FUNCTION_BLOCK TcoDigitalSensor EXTENDS TcoCore.TcoComponent
VAR_IN_OUT
	inoSignal : BOOL;
END_VAR

VAR
	_signal : BOOL;
	_adr : ULINT;
END_VAR

IF(__ISVALIDREF(inoSignal)) THEN
	_signal := inoSignal;
	_adr := ADR(inoSignal);
END_IF;

METHOD FB_init : BOOL
VAR_INPUT
	bInitRetains : BOOL; // if TRUE, the retain variables are initialized (warm start / cold start)
	bInCopyCode : BOOL;  // if TRUE, the instance afterwards gets moved into the copy code (online change)
	Parent : ITcoObject;
END_VAR
END_METHOD

{attribute 'monitoring' := 'variable'}
PROPERTY IsFalse : BOOL
GET
IsFalse := NOT _signal;
Messenger.Info('Expecting `negative` signal');
END_GET
END_PROPERTY

{attribute 'monitoring' := 'variable'}
PROPERTY IsTrue : BOOL
GET
IsTrue := _signal;
Messenger.Info('Expecting `positive` signal');
END_GET
END_PROPERTY

(*~
	<docu>
		<summary>
			Restores this instance to the Ready state. Can be called explicitly or from within one of the restore mechanisms.	
		</summary>			
	</docu>	
~*)
METHOD  Restore : ITcoRestorable
// No implementation needed for this componet.
END_METHOD

(*~
	<docu>
		<summary>
		    Custom service (manual, maintenance) logic.
			This method must be implemented in derived class.
		</summary>			
	</docu>	
~*)
METHOD PROTECTED  ServiceMode
END_METHOD

END_FUNCTION_BLOCK

(* stored: Version 1.1.0.1, ProductVersion 3.1.4024.6
   POU TcoDigitalSensor: Id {940ec0d0-0377-0ad5-2841-be1fc78a02da}, SpecialFunc None
   Method FB_init: Id {ab66c675-5325-0f32-2184-6fc98948f748}
   Property IsFalse: Id {48e6cf82-019c-09fc-0b62-4318a8025ee4}
   Get Get: Id {c23c2e72-5cf6-0203-23ee-9d8001c6afd4}
   Property IsTrue: Id {c588e641-6ea7-04c2-2aae-c7227089c8ae}
   Get Get: Id {2089a10e-bba5-06e8-1e33-1a25b4fcfa09}
   Method Restore: Id {19478393-8665-053e-2aa6-99986ee029e0}
   Method ServiceMode: Id {27fb8047-ad11-0e35-19c9-b36842b34792} *)
